{attribute 'qualified_only'}
VAR_GLOBAL CONSTANT
	nPytmcTypesArrayLength : UINT := 99;
END_VAR

(* stored: Version 1.1.0.1, ProductVersion 3.1.4026.12
   GVL GVL: Id {4625bf49-36db-4e2a-9d02-8d0b19f122e5} *)
